// TIA Portal V19 export
TYPE "MatCountData"
// stored: Access Published
   STRUCT
      Standstill { ExternalVisible := 'False'; ExternalWritable := 'False'} : Bool;
      CounterValid { ExternalVisible := 'False'; ExternalWritable := 'False'} : Bool;
      AxPosition { ExternalVisible := 'False'; ExternalWritable := 'False'} : LReal;
      AxPositionPrevious { ExternalVisible := 'False'; ExternalWritable := 'False'} : LReal;
      FAK { ExternalVisible := 'False'; ExternalWritable := 'False'} : LReal;
      CounterValueInit { ExternalVisible := 'False'; ExternalWritable := 'False'} : LReal;
      CounterOffset { ExternalVisible := 'False'; ExternalWritable := 'False'} : LReal;
      CounterValue { ExternalWritable := 'False'} : LReal;
      FAKPrevious { ExternalVisible := 'False'; ExternalWritable := 'False'} : LReal;
      AX_MODULE { ExternalVisible := 'False'; ExternalWritable := 'False'} : LReal;
      COUNTER_MODULE { ExternalVisible := 'False'; ExternalWritable := 'False'} : LReal;
   END_STRUCT;
END_TYPE
